// TIA Portal V15.1 export
// export: Created 2024-05-17T05:38:40.1002295Z, ExportSetting WithDefaults, DisplayName Totally Integrated Automation Portal, DisplayVersion V15.1 Update 5, DisplayName TIA Portal Openness, DisplayVersion V15.1 Update 5, DisplayName SINAMICS Startdrive Advanced, DisplayVersion V15.1, DisplayName G130, G150, S120, S150, SINAMICS MV, S210, DisplayVersion V15.1, DisplayName G110M, G120, G120C, G120D, G120P, DisplayVersion V15.1, DisplayName STEP 7 Professional, DisplayVersion V15.1 Update 5, DisplayName STEP 7 Safety, DisplayVersion V15.1, DisplayName WinCC Professional, DisplayVersion V15.1 Update 5, DisplayName SIMATIC Visualization Architect, DisplayVersion V15.1
FUNCTION_BLOCK "LGBCrossConvStopHighSpeed"   // FB6708, FBD
TITLE = LGBCrossConvStopHighSpeed
{ S7_Optimized_Access := 'TRUE' }
VERSION : 0.1
// stored: AutoNumber false, IsIECCheckEnabled false, IsRetainMemResEnabled false, MemoryReserve 100, SetENOAutomatically False, UDAEnableTagReadback false
   VAR_INPUT
      I_StopHighSpeedDet { ExternalAccessible := 'False'; ExternalVisible := 'False'; ExternalWritable := 'False'} : Bool;   // Stop High Speed detection
      I_AllDet { ExternalAccessible := 'False'; ExternalVisible := 'False'; ExternalWritable := 'False'} : Bool;   // AND of all detections
      I_TrfInCmd { ExternalAccessible := 'False'; ExternalVisible := 'False'; ExternalWritable := 'False'} : Bool;   // Transfer In Command Cross movement
   END_VAR
   VAR_OUTPUT
      O_StopHighSpeed { ExternalAccessible := 'False'; ExternalVisible := 'False'; ExternalWritable := 'False'} : Bool;   // Stop High Speed
      O_StopHighSpeedDet { ExternalAccessible := 'False'; ExternalVisible := 'False'; ExternalWritable := 'False'} : Bool;   // The Stop High Speed detection was activated during transfer (Cross movement)
   END_VAR
   VAR_IN_OUT
      IO_Modes : "Modes";   // Modes
      H_ManSelMovFromOtherCC { ExternalAccessible := 'False'; ExternalVisible := 'False'; ExternalWritable := 'False'} : Bool;   // HMI Command, transfer from other Cross Conveyor / HMI Command
      IO_ModesOtherCC : "Modes";   // Modes / Modes Cross Conveyor Y
   END_VAR
   VAR RETAIN
      "Stop High Speed" { ExternalAccessible := 'False'; ExternalVisible := 'False'; ExternalWritable := 'False'} : Bool;   // Stop High Speed
      StopHighSpeedDetActivated { ExternalAccessible := 'False'; ExternalVisible := 'False'; ExternalWritable := 'False'} : Bool;   // The Stop High Speed detection was activated during transfer (Cross movement)
   END_VAR
BEGIN

REGION Network 1: **** 5.2 - Equations - Flow **** The Stop High Speed detection was activated during transfer (Cross movement)
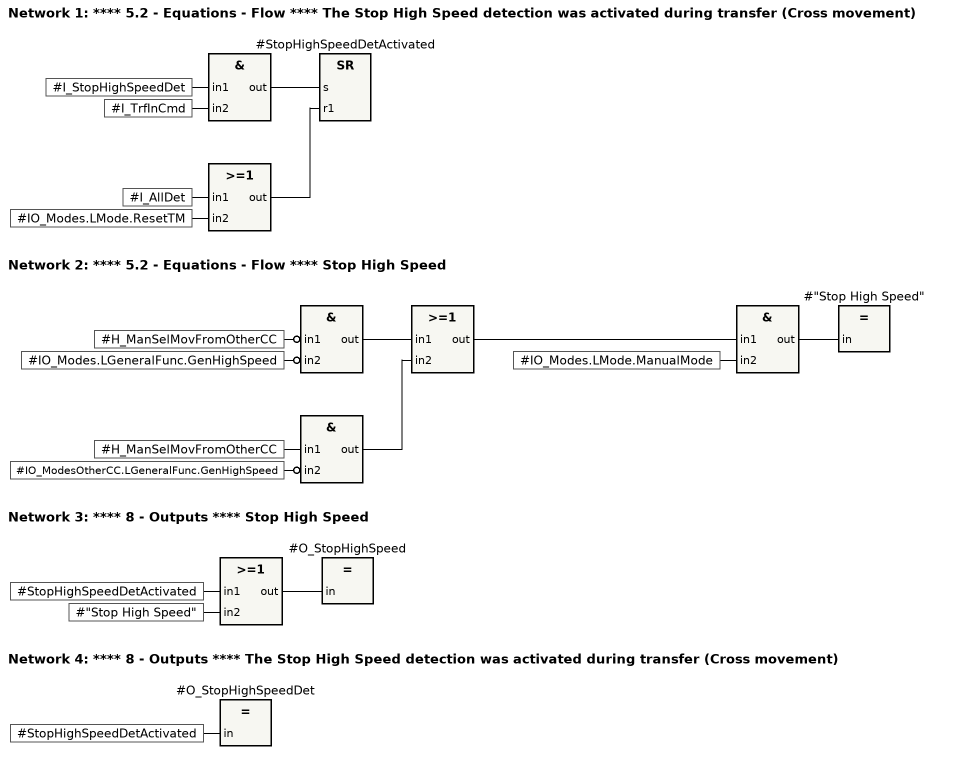
   IF #I_StopHighSpeedDet AND #I_TrfInCmd THEN
       #StopHighSpeedDetActivated := TRUE;   // SR flip-flop
   END_IF;
   IF #I_AllDet OR #IO_Modes.LMode.ResetTM THEN #StopHighSpeedDetActivated := FALSE; END_IF;
END_REGION

REGION Network 2: **** 5.2 - Equations - Flow **** Stop High Speed
   #"Stop High Speed" := ((NOT #H_ManSelMovFromOtherCC AND NOT #IO_Modes.LGeneralFunc.GenHighSpeed) OR (#H_ManSelMovFromOtherCC AND NOT #IO_ModesOtherCC.LGeneralFunc.GenHighSpeed)) AND #IO_Modes.LMode.ManualMode;
END_REGION

REGION Network 3: **** 8 - Outputs **** Stop High Speed
   #O_StopHighSpeed := #StopHighSpeedDetActivated OR #"Stop High Speed";
END_REGION

REGION Network 4: **** 8 - Outputs **** The Stop High Speed detection was activated during transfer (Cross movement)
   #O_StopHighSpeedDet := #StopHighSpeedDetActivated;
END_REGION
END_FUNCTION_BLOCK
